# EPICS StreamDevice protocol: lvremoteSup/lvremote_string.proto
Terminator = CR LF;
path="%#/\//\\/";

ReadTimeout = 20;
WriteTimeout = 200;
ReplyTimeout = 100;
LockTimeout = 5000;

getString {
    out "LVGET \${1}" ${path} ",\$2";
    in "%#s";
}
sendString {
    out "LVPUT \$1" ${path} ",\$2,%s";
    @init { getString; }
}
